// TIA Portal V20 export
VAR_GLOBAL   // PLC tag table "LConSMC_Errors"
END_VAR
VAR_GLOBAL CONSTANT   // user constants
   LCON_ERROR_RFG_INVALID_CYCLE_TIME : DWord := 16#1106_8001;   // Function block is not called in a cylic OB (cycle time = 0.0)
   LCON_ERROR_SECTIONAL_DRIVE_DATA_ADAPTION : DWord := 16#7102_8009;   // Error during data adaption of the TO
   LCON_ERROR_ENABLE_INTERFACE_ADDITIVE_TORQUE : DWord := 16#3107_8004;   // Error MC command MC_AdditiveTorque. ErrorID of MC command is displayed at output "subfunctionState" of FB LConSMC_EnableInterface
   LCON_ERROR_WINDER_INVALID_DIAMETER_MODE : DWord := 16#5105_800B;   // Position based diameter calculation mode can't be used for speed axes
   LCON_ERROR_ENABLE_INTERFACE_HALT : DWord := 16#3107_800E;   // Error MC command MC_Halt. ErrorID of MC command is displayed at output "subfunctionState" of FB LConSMC_EnableInterface
   LCON_ERROR_INTEGRATOR_INVALID_CYCLE_TIME : DWord := 16#1102_8001;   // Function block is not called in a cylic OB (cycle time = 0.0)
   LCON_ERROR_DIFFERENTIATOR_INVALID_CYCLE_TIME : DWord := 16#1103_8001;   // Function block is not called in a cylic OB (cycle time = 0.0)
   LCON_ERROR_SECTIONAL_DRIVE_DRIVE_NOT_ENABLED : DWord := 16#7102_8010;   // The drive must be enabled when enabling the function block
   LCON_ERROR_CALC_TARGET_DIAM_STOP_COND_INVALID_CYCLE_TIME : DWord := 16#4004_8001;   // Function block is not called in a cylic OB (cycle time = 0.0)
   LCON_ERROR_WINDER_INVALID_TYPE_OF_AXIS : DWord := 16#5105_800A;   // Invalid axis type selected
   LCON_ERROR_DIAM_CALC_MAX_BUFFER_SIZE : DWord := 16#5104_8006;   // The maximum buffer size for the floating diameter calculation has been exceeded. Reduce the "measuringRevolutionCount" or increase the "diameterOutputRate"
   LCON_ERROR_WINDER_DATA_ADAPTION : DWord := 16#5105_8009;   // Error during data adaption of the TO
   LCON_ERROR_DT1_INVALID_CYCLE_TIME : DWord := 16#1104_8001;   // Function block is not called in a cylic OB (cycle time = 0.0)
   LCON_ERROR_TORQUE_PRECONTROL_INVALID_INPUT : DWord := 16#6101_8008;   // diameter <= 0.0
   LCON_ERROR_PT1_INVALID_CYCLE_TIME : DWord := 16#1101_8001;   // Function block is not called in a cylic OB (cycle time = 0.0)
   LCON_ERROR_SECTIONAL_DRIVE_INVALID_TYPE_OF_AXIS : DWord := 16#7102_800A;   // Invalid axis type selected
   LCON_ERROR_WINDER_INVALID_CYCLE_TIME : DWord := 16#5105_8001;   // Function block is not called in a cylic OB (cycle time = 0.0)
   LCON_ERROR_FRICTION_V2_MOVE_VELOCITY : DWord := 16#3113_8601;   // Error MC command MC_MoveVelocity. ErrorID of MC command is displayed at FB output "subfunctionState"
   LCON_ERROR_DIAM_CALC_INVALID_MODE : DWord := 16#5104_800B;   // Invalid diameter calculation mode selected ( < 0 or > 5)
   LCON_ERROR_KP_ADAPTION_TELEGRAM_EXTENSION : DWord := 16#3109_8002;   // Invalid telegram address: * No valid HW-Address connected * Invalid telegram length (Must be at least two Bytes)
   LCON_ERROR_WINDER_DRIVE_NOT_ENABLED : DWord := 16#5105_8010;   // The drive must be enabled when enabling the function block
   LCON_ERROR_WI_TORQUE_PRECONTROL_INVALID_CYCLE_TIME : DWord := 16#4102_8001;   // Function block is not called in a cylic OB (cycle time = 0.0)
   LCON_ERROR_ENABLE_INTERFACE_MOVE_VELOCITY : DWord := 16#3107_800C;   // Error MC command MC_MoveVelocity. ErrorID of MC command is displayed at output "subfunctionState" of FB LConSMC_EnableInterface
   LCON_ERROR_RFGJ_INVALID_CYCLE_TIME : DWord := 16#1107_8001;   // Function block is not called in a cylic OB (cycle time = 0.0)
   LCON_ERROR_ANALOG_INPUT_INVALID_CYCLE_TIME : DWord := 16#1109_8001;   // Function block is not called in a cylic OB (cycle time = 0.0)
   LCON_ERROR_DIAM_CALC_INVALID_CYCLE_TIME : DWord := 16#5104_8001;   // Function block is not called in a cylic OB (cycle time = 0.0)
   LCON_ERROR_SECTIONAL_DRIVE_INVALID_CYCLE_TIME : DWord := 16#7102_8001;   // Function block is not called in a cylic OB (cycle time = 0.0)
   LCON_ERROR_CALC_TARGET_DIAM_STOP_COND_INVALID_CONFIGURATION : DWord := 16#4004_8000;   // Invalid configuration data: * windingMode < 0 * windinMode > 1 * minDiameter >= maxDiameter * rampUpTime <= 0.0 * ramDownTime <= 0.0 * roundingTIme <= 0.0
   LCON_ERROR_PID_INVALID_CYCLE_TIME : DWord := 16#1105_8001;   // Function block is not called in a cylic OB (cycle time = 0.0)
   LCON_ERROR_WI_TORQUE_PRECONTROL_INVALID_INPUT : DWord := 16#4102_8008;   // Invalid input data: * diamActVal <= 0 * diamActVal < diamMin
   LCON_ERROR_TAPER_INVALID_INPUT : DWord := 16#4101_8008;   // Invalid input data: * diamActVal <= 0 for taperMode <> 0 * taperMode < 0 * taperMode > 4
   LCON_ERROR_TABLE_CHAR_ENTRIES_NOT_MONOTONIC : DWord := 16#0106_8007;   // The table entries are not monotonic increasing/decreasing
   LCON_ERROR_ENABLE_INTERFACE_TORQUE_RANGE : DWord := 16#3107_8005;   // Error MC command MC_TorqueRange. ErrorID of MC command is displayed at output "subfunctionState" of FB LConSMC_EnableInterface
   LCON_ERROR_DIAM_CALC_INVALID_CONFIGURATION : DWord := 16#5104_8000;   // Invalid configuration data for diameter calculation: * minDia/maxDia <= 0.0 * minDia > maxDia * diameterFilterTime < 0.0 * webThickness <= 0.0 (if mode 1/4 selected) * typeOfWinder < 0 or > 3 * measuringRevolutionCount <= 0.0 * measuringRevolutionCount < diameterOutputRate
   LCON_ERROR_WINDER_INVALID_CONFIGURATION : DWord := 16#5105_8000;   // Invalid configuration data for winder: * Invalid axis unit * controlMode < 0 or > 5 * typeOfWinder < 0 or > 3 * diameter calculation mode < 0 or > 5 * gearRatio <= 0 * No telegram 750 connected for torque controlled modes * diamConfig.minDia/maxDia = 0.0 * diamConfig.minDia > diamConfig.maxDia
   LCON_ERROR_TAPER_INVALID_CONFIGURATION : DWord := 16#4101_8000;   // Invalid configuration data for tension taper: * taperMode < 0 or > 4 * upperLimitTaper < lowerLimitTaper * lowerLimitTaper < 0.0 Additionally for taperMode 1-3: * taperDiameterStart < 0.0 * taperDiameterMax <= taperDiameterStart * taperRatio < 0.0 * taperRatio > 100.0
   LCON_ERROR_TABLE_CHAR_INVALID_CONFIGURATION : DWord := 16#0106_8000;   // Invalid configuration data for TableChar: * sizeOfArray < 2 * sizeOfArray > 20
   LCON_ERROR_FRICTION_V2_INVALID_CONFIGURATION : DWord := 16#3113_8000;   // Invalid configuration data for friction measurement: * sizeOfArray < 1 * No telegram 750 active at TO * The speed setpoints (speedValues) are not increasing * A linear axis has been connected
   LCON_ERROR_CALC_STOP_DISTANCE_INVALID_CONFIGURATION : DWord := 16#0005_8000;   // Invalid configuration data for CalcStopDistance: * maxVelocity = 0.0 * rampDownTime = 0.0 * (roundingTime <> 0.0 and rampUpTime = 0.0)
   LCON_ERROR_PID_INVALID_CONFIGURATION : DWord := 16#1105_8000;   // Invalid configuration data for PID controller: * lowerLimit > upperLimit
   LCON_ERROR_RFG_INVALID_CONFIGURATION : DWord := 16#1106_8000;   // Invalid configuration data for RFG: * rampTimeMode < 0 * rampTimeMode > 1
   LCON_ERROR_TORQUE_PRECONTROL_INVALID_CONFIGURATION : DWord := 16#6101_8000;   // Invalid configuration data for sectional drive torque precontrol: * JFix/JMandrel/JMot < 0.0 * 0 < typeOfDrive > 1
   LCON_ERROR_AVARAGE_INVALID_CONFIGURATION : DWord := 16#0105_8000;   // Invalid configuration data for AverageValue calculation: * sizeOfArray < 2 * sizeOfArray > 20
   LCON_ERROR_TPID_INVALID_CONFIGURATION : DWord := 16#1108_8000;   // Invalid configuration data for TPID controller: * setNominalValue <= 0.0
   LCON_ERROR_ANALOG_INPUT_INVALID_CONFIGURATION : DWord := 16#1109_8000;   // Invalid configuration data for AnalogInput: * base = 0.0
   LCON_ERROR_KP_ADAPTION_INVALID_CONFIGURATION : DWord := 16#3109_8000;   // Invalid configuration data for Kp Adaption: * diamConfig.maxDia = 0.0 * diamConfig.maxDia <= diamConfig.minDia * diameter <= 0.0 * torquePreControl.maxInertia <= 0.0 * torquePreControlDiag.totalInertia <= 0.0
   LCON_ERROR_WI_TORQUE_PRECONTROL_INVALID_CONFIGURATION : DWord := 16#4102_8000;   // Invalid configuration data for winder torque precontrol: * gearRatio/diamMin/fillFactor <= 0.0 * density/width/JFix/JMandrel/JMot < 0.0 * diamMax <= diamMin * typeOfWinder < 0 or > 3
   LCON_ERROR_RFGJ_INVALID_CONFIGURATION : DWord := 16#1107_8000;   // Invalid configuration data for RFGJ: * rampTimeMode < 0 * rampTimeMode > 1 * nominalValue = 0.0
   LCON_ERROR_SECTIONAL_DRIVE_INVALID_CONFIGURATION : DWord := 16#7102_8000;   // Invalid configuration data for sectional drive: * Invalid axis unit * controlMode < 0 or > 5 * typeOfDrive < 0 or > 1 * sectionalConfig.diameter <= 0.0 * gearRatio <= 0 * No telegram 750 connected for torque controlled modes
   LCON_ERROR_FRICTION_INVALID_CONFIGURATION : DWord := 16#3103_8000;   // Invalid configuration data for friction measurement: * sizeOfArray < 1
   LCON_ERROR_CALC_TENSION_INVALID_INPUTS : Word := 16#0000_8200;   // Invalid input data: * gearRatio <= 0.0 * diameter <= 0.0
   LCON_ERROR_ENABLE_INTERFACE_INVALID_AXIS : DWord := 16#3107_8006;   // Invalid axis connected to function block. Only TO_SpeedAxis, TO_PositioningAxis or TO_SynchronousAxis are supported
   LCON_ERROR_ENABLE_INTERFACE_MOVE_ABORTED : DWord := 16#3107_8007;   // Error MC command MC_MoveVelocity. The internal move command has been aborted from an external command. The axis will be stopped
   LCON_ERROR_CALC_TENSION_INVALID_STATE : Word := 16#0000_8201;   // Internal error: Invalid state
   LCON_ERROR_ENABLE_INTERFACE_INVALID_STATE : DWord := 16#3107_8600;   // Internal error: Invalid state
END_VAR
